FUNCTION_BLOCK FB_ExDevUML_SM
VAR_INPUT
END_VAR
VAR_OUTPUT
END_VAR
VAR
END_VAR

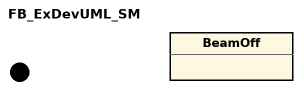
STATECHART FB_ExDevUML_SM  // abortable
    START StartState1
    STATE BeamOff
END_STATECHART

END_FUNCTION_BLOCK

(* stored: Version 1.1.0.1, ProductVersion 3.1.4022.10
   POU FB_ExDevUML_SM: Id {0d23ae89-ec70-4541-86b1-c25e855b3f6c}, SpecialFunc None *)
